{attribute 'GeneratedUsingTerminal: EL5032-0000-0021'}
{attribute addProperty BoxType "EL5032-0000-0021"}
{attribute addProperty Description "EL5032 2Ch. EnDat Encoder"}
{attribute addProperty Physics "KK"}
{attribute addProperty Id "FB_Inputs_Channel_1AT %I*FB_Inputs_Channel_7405098814FB_Inputs_Channel_2AT %I*FB_Inputs_Channel_7405098814WcStateAT %I*WcState_9091E0EB2InfoDataAT %I*InfoData_32EB74EA10"}
{attribute addProperty CRC "1814315440"}
{attribute addProperty Size "40"}
TYPE EL5032_6C2441B0 EXTENDS EtcSlaveTerminalBase_947E5A46 :
STRUCT
	{attribute addProperty Name "FB_Inputs_Channel_1"}
	FB_Inputs_Channel_1 : FB_Inputs_Channel_74050988;
	{attribute addProperty Name "FB_Inputs_Channel_2"}
	FB_Inputs_Channel_2 : FB_Inputs_Channel_74050988;
	{attribute addProperty Name "WcState"}
	WcState : WcState_9091E0EB;
	{attribute addProperty Name "InfoData"}
	InfoData : InfoData_32EB74EA;
END_STRUCT
END_TYPE

(* stored: Version 1.2.0.0, ProductVersion 3.1.4024.9
   DUT EL5032_6C2441B0: Id {1a2aa42f-4a4e-461b-b769-118b34c9e191} *)
